// TIA Portal project "practical4 simba chipsFINAL" (V16)

(* hardware
DEVICE "S7300/ET200M station_1"  S7-300 station
   slot 0: "Rail_0"  Rail  6ES7 390-1***0-0AA0
   slot 1: "PS 307 2A_1"  PS 307 2A  6ES7 307-1BA01-0AA0
   slot 2: "PLC_1"  CPU 314C-2 DP  6ES7 314-6CH04-0AB0  V3.3
      slot 0: "MPI interface_1"  MPI
      slot 1: "DP interface_1"  DP
      slot 2: "DI 24/DO 16_1"  DI24/DO16
      slot 3: "AI 5/AO 2_1"  AI5/AO2
      slot 4: "Count_1"  Counter
      slot 5: "Positioning_1"  Positioning
DEVICE "HMI_1"  KTP700 Basic DP
   slot 0: "HMI_1"  KTP700 Basic DP  6AV2 123-2GA03-0AX0  16.0.0.0
   slot 1: "HMI_RT_1"  KTP700 Basic DP  6AV2 123-2GA03-0AX0  16.0.0.0
   slot 7: "HMI_1.MPI/DP_CP_1"  MPI/DP Interface  16.0.0.0
*)

// ===== PLC "PLC_1"  CPU 314C-2 DP =====

VAR_GLOBAL   // PLC tag table "Default tag table"
   "START" AT %M0.0 : Bool;
   "STOP" AT %M0.1 : Bool;
   "CONVEYOR 4" AT %Q0.0 : Bool;
   "RUNMODE" AT %Q1.3 : Bool;
   "OIL HEATER" AT %Q0.1 : Bool;
   "OIL HEATER TIMER" AT %T0 : Timer;
   "HEATER OUTPUT" AT %Q0.2 : Bool;
   "CONVEYOR 1" AT %Q0.3 : Bool;
   "CUTTING MACHINE" AT %Q0.4 : Bool;
   "CONVEYOR 2" AT %Q0.5 : Bool;
   "FRYING MACHINE" AT %Q0.6 : Bool;
   "CHIPS FRIER" AT %T1 : Timer;
   "CONVEYOR 3" AT %Q0.7 : Bool;
   "SENSOR" AT %M0.3 : Bool;
   "CHIPS COUNTER" AT %C0 : Counter;
   "COUNTER OUTPUT" AT %Q1.0 : Bool;
   "RESET" AT %M0.4 : Bool;
   "MAX" AT %MW0 : Word;
   "LOADING DURATION" AT %Q1.1 : Bool;
   "LOADING TIMER" AT %T2 : Timer;
   "TRUCK" AT %Q1.2 : Bool;
   "DELAY CONVEYOR 2" AT %T3 : Timer;
   "COMPARATOR OUTPUT" AT %Q1.4 : Bool;
   "SET VALUE" AT %M0.5 : Bool;
END_VAR

ORGANIZATION_BLOCK "Main"   // OB1, LAD
TITLE = "Main Program Sweep (Cycle)"
{ S7_Optimized_Access := 'FALSE' }
VERSION : 0.1
   VAR_TEMP
      OB1_EV_CLASS : Byte;   // Bits 0-3 = 1 (Coming event), Bits 4-7 = 1 (Event class 1)
      OB1_SCAN_1 : Byte;   // 1 (Cold restart scan 1 of OB 1), 3 (Scan 2-n of OB 1)
      OB1_PRIORITY : Byte;   // Priority of OB Execution
      OB1_OB_NUMBR : Byte;   // 1 (Organization block 1, OB1)
      OB1_RESERVED_1 : Byte;   // Reserved for system
      OB1_RESERVED_2 : Byte;   // Reserved for system
      OB1_PREV_CYCLE : Int;   // Cycle time of previous OB1 scan (milliseconds)
      OB1_MIN_CYCLE : Int;   // Minimum cycle time of OB1 (milliseconds)
      OB1_MAX_CYCLE : Int;   // Maximum cycle time of OB1 (milliseconds)
      OB1_DATE_TIME : Date_And_Time;   // Date and time OB1 started
   END_VAR
   VAR_TEMP   // added for the SCL form of the ladder/FBD networks
      _w1 : Bool;
      _s5time1 : S5Time;
   END_VAR
BEGIN

REGION Network 1: LATCHING CIRCUIT
   // Start button activates the system, Stop button deactivates the system. Runnmode is used as holding switch.
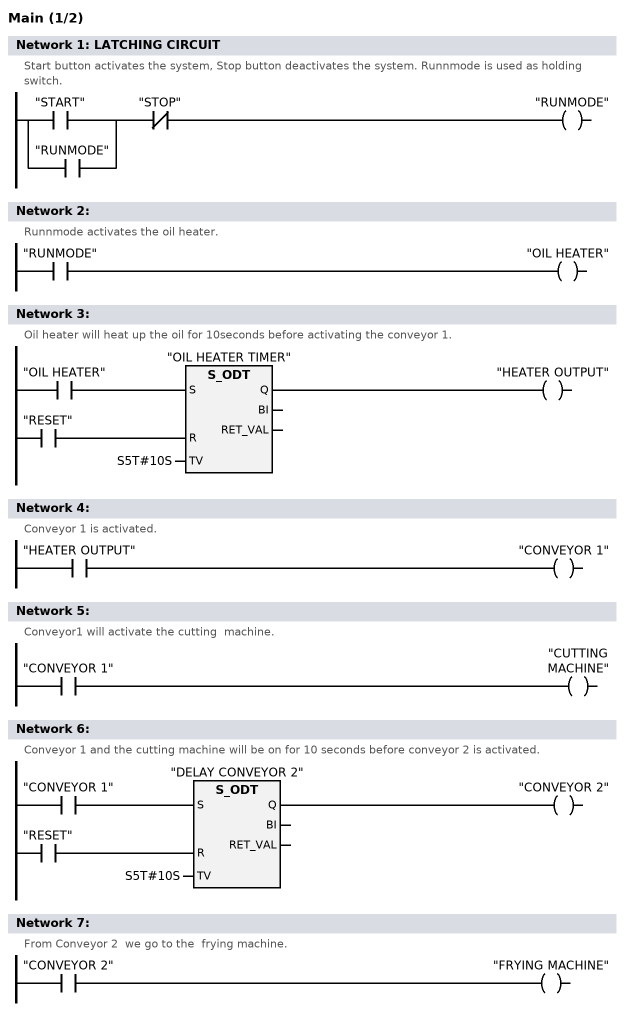
   RUNG wire#powerrail
      Contact( "START" )
      wire#w1
      I_Contact( "STOP" )
      Coil( "RUNMODE" )
   END_RUNG
   RUNG wire#powerrail
      Contact( "RUNMODE" )
   END_RUNG wire#w1
   // the same network as SCL:
   "RUNMODE" := ("START" OR "RUNMODE") AND NOT "STOP";
END_REGION

REGION Network 2
   // Runnmode activates the oil heater.
   RUNG wire#powerrail
      Contact( "RUNMODE" )
      Coil( "OIL HEATER" )
   END_RUNG
   // the same network as SCL:
   "OIL HEATER" := "RUNMODE";
END_REGION

REGION Network 3
   // Oil heater will heat up the oil for 10seconds before activating the conveyor 1.
   RUNG wire#powerrail
      Contact( "OIL HEATER" )
      S_ODT(T_NO := "OIL HEATER TIMER", R := wire#w1, TV := S5T#10S, BI =>, RET_VAL =>)
      Coil( "HEATER OUTPUT" )
   END_RUNG
   RUNG wire#powerrail
      Contact( "RESET" )
   END_RUNG wire#w1
   // the same network as SCL:
   #_s5time1 := S_ODT(T_NO := "OIL HEATER TIMER", S := "OIL HEATER", R := "RESET", TV := S5T#10S, Q => #_w1);
   "HEATER OUTPUT" := #_w1;
END_REGION

REGION Network 4
   // Conveyor 1 is activated.
   RUNG wire#powerrail
      Contact( "HEATER OUTPUT" )
      Coil( "CONVEYOR 1" )
   END_RUNG
   // the same network as SCL:
   "CONVEYOR 1" := "HEATER OUTPUT";
END_REGION

REGION Network 5
   // Conveyor1 will activate the cutting  machine.
   RUNG wire#powerrail
      Contact( "CONVEYOR 1" )
      Coil( "CUTTING MACHINE" )
   END_RUNG
   // the same network as SCL:
   "CUTTING MACHINE" := "CONVEYOR 1";
END_REGION

REGION Network 6
   // Conveyor 1 and the cutting machine will be on for 10 seconds before conveyor 2 is activated.
   RUNG wire#powerrail
      Contact( "CONVEYOR 1" )
      S_ODT(T_NO := "DELAY CONVEYOR 2", R := wire#w1, TV := S5T#10S, BI =>, RET_VAL =>)
      Coil( "CONVEYOR 2" )
   END_RUNG
   RUNG wire#powerrail
      Contact( "RESET" )
   END_RUNG wire#w1
   // the same network as SCL:
   #_s5time1 := S_ODT(T_NO := "DELAY CONVEYOR 2", S := "CONVEYOR 1", R := "RESET", TV := S5T#10S, Q => #_w1);
   "CONVEYOR 2" := #_w1;
END_REGION

REGION Network 7
   // From Conveyor 2  we go to the  frying machine.
   RUNG wire#powerrail
      Contact( "CONVEYOR 2" )
      Coil( "FRYING MACHINE" )
   END_RUNG
   // the same network as SCL:
   "FRYING MACHINE" := "CONVEYOR 2";
END_REGION

REGION Network 8
   // Frying machine will fry the chips for 20 seconds  before transporting  the chips via conveyor 3 to the boxes.
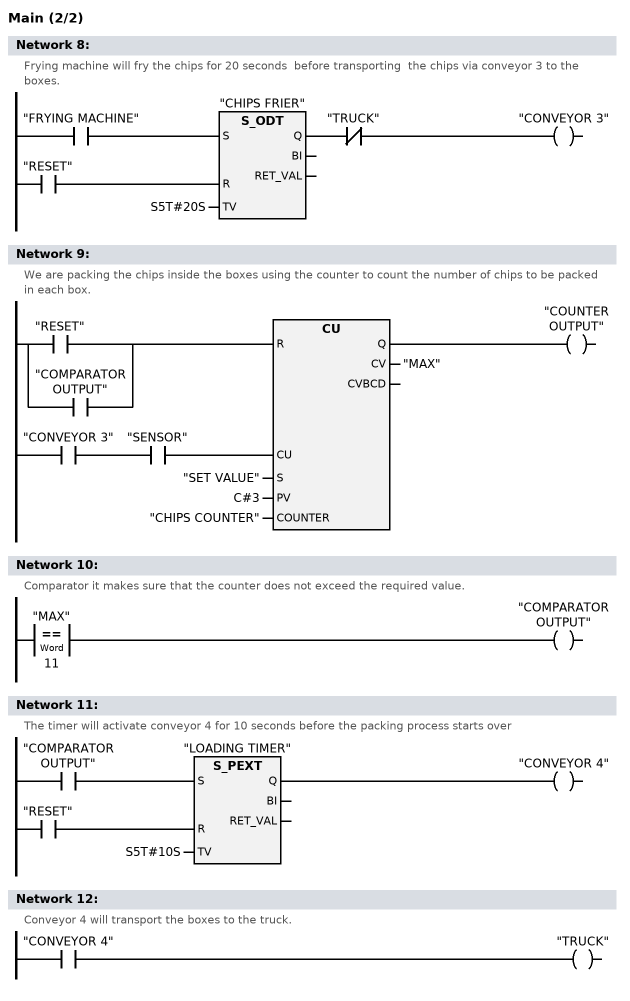
   RUNG wire#powerrail
      Contact( "FRYING MACHINE" )
      S_ODT(T_NO := "CHIPS FRIER", R := wire#w1, TV := S5T#20S, BI =>, RET_VAL =>)
      I_Contact( "TRUCK" )
      Coil( "CONVEYOR 3" )
   END_RUNG
   RUNG wire#powerrail
      Contact( "RESET" )
   END_RUNG wire#w1
   // the same network as SCL:
   #_s5time1 := S_ODT(T_NO := "CHIPS FRIER", S := "FRYING MACHINE", R := "RESET", TV := S5T#20S, Q => #_w1);
   "CONVEYOR 3" := #_w1 AND NOT "TRUCK";
END_REGION

REGION Network 9
   // We are packing the chips inside the boxes using the counter to count the number of chips to be packed  in each box.
   // no SCL statement known for Cu: written as a call
   Cu(cu := "CONVEYOR 3" AND "SENSOR",
      r := "RESET" OR "COMPARATOR OUTPUT",
      s := "SET VALUE",
      pv := C#3,
      "counter" := "CHIPS COUNTER",
      q => #_w1,
      cv => "MAX");
   "COUNTER OUTPUT" := #_w1;
END_REGION

REGION Network 10
   // Comparator it makes sure that the counter does not exceed the required value.
   RUNG wire#powerrail
      { S7_Templates := "SrcType := Word" } EQ_Contact(in1 := "MAX", in2 := 11)
      Coil( "COMPARATOR OUTPUT" )
   END_RUNG
   // the same network as SCL:
   "COMPARATOR OUTPUT" := "MAX" = 11;
END_REGION

REGION Network 11
   // The timer will activate conveyor 4 for 10 seconds before the packing process starts over
   RUNG wire#powerrail
      Contact( "COMPARATOR OUTPUT" )
      S_PEXT(T_NO := "LOADING TIMER", R := wire#w1, TV := S5T#10S, BI =>, RET_VAL =>)
      Coil( "CONVEYOR 4" )
   END_RUNG
   RUNG wire#powerrail
      Contact( "RESET" )
   END_RUNG wire#w1
   // the same network as SCL:
   #_s5time1 := S_PEXT(T_NO := "LOADING TIMER",
                       S := "COMPARATOR OUTPUT",
                       R := "RESET",
                       TV := S5T#10S,
                       Q => #_w1);
   "CONVEYOR 4" := #_w1;
END_REGION

REGION Network 12
   // Conveyor 4 will transport the boxes to the truck.
   RUNG wire#powerrail
      Contact( "CONVEYOR 4" )
      Coil( "TRUCK" )
   END_RUNG
   // the same network as SCL:
   "TRUCK" := "CONVEYOR 4";
END_REGION
END_ORGANIZATION_BLOCK

(* ===== HMI "HMI_RT_1" =====
system functions are stored by id; their names below are inferred from use
connection "HMI_Connection_1": IF1 B, SIMATIC S7 300/400 MPI

HMI tags "Default tag table"
   "Tag_ScreenNumber" : UInt, internal
   "START" : Bool = PLC START AT %M0.0, 1 s
   "STOP" : Bool = PLC STOP AT %M0.1, 1 s
   "SENSOR" : Bool = PLC SENSOR AT %M0.3, 1 s
   "OIL HEATER" : Bool = PLC "OIL HEATER" AT %Q0.1, 1 s
   "HEATER OUTPUT" : Bool = PLC "HEATER OUTPUT" AT %Q0.2, 1 s
   "CONVEYOR 2" : Bool = PLC "CONVEYOR 2" AT %Q0.5, 1 s
   "CONVEYOR 1" : Bool = PLC "CONVEYOR 1" AT %Q0.3, 1 s
   "CUTTING MACHINE" : Bool = PLC "CUTTING MACHINE" AT %Q0.4, 1 s
   "OIL HEATER TIMER" : Timer = PLC "OIL HEATER TIMER" AT %T0, 1 s
   "RUNMODE" : Bool = PLC RUNMODE AT %Q1.3, 1 s
   "DELAY CONVEYOR 2" : Timer = PLC "DELAY CONVEYOR 2" AT %T3, 1 s
   "CONVEYOR 3" : Bool = PLC "CONVEYOR 3" AT %Q0.7, 1 s
   "FRYING MACHINE" : Bool = PLC "FRYING MACHINE" AT %Q0.6, 1 s
   "COUNTER OUTPUT" : Bool = PLC "COUNTER OUTPUT" AT %Q1.0, 1 s
   "CHIPS FRIER" : Timer = PLC "CHIPS FRIER" AT %T1, 1 s
   "CHIPS COUNTER" : Counter = PLC "CHIPS COUNTER" AT %C0, 1 s
   "CONVEYOR 4" : Bool = PLC "CONVEYOR 4" AT %Q0.0, 1 s
   "movement" : Int, internal
   "LOADING DURATION" : Bool = PLC "LOADING DURATION" AT %Q1.1, 1 s
   "LOADING TIMER" : Timer = PLC "LOADING TIMER" AT %T2, 1 s
   "RESET" : Bool = PLC RESET AT %M0.4, 1 s

Template "Template_1" 800x480
   SymbolicIOField "Symbolic_IO_Field_Screen" at 93,9 size 600x33; TextOff '0'; TextOn '1'; TextList "TextList_ScreenNames"
      ProcessValue <- "Tag_ScreenNumber"
      on Change: ActivateScreenByNumber("Tag_ScreenNumber", 0)
   DateTimeField "HmiScreenItemData" at 695,25 size 105x25
   DateTimeField "HmiScreenItemData_1" at 695,0 size 105x25
   GraphicView "Logo" at 0,0 size 91x51; Picture "Logo of HMI_1"

screen "Root screen" 800x480, template "Template_1"
   on GenerateScreen: function_f9c01323("movement", 1, 100, 0, 1)
   TextField "HmiScreenItemData" at 43,19 size 640x25; Text 'Welcome to HMI_1 (KTP700 Basic+ DP)!'
   Button "Button_1" at 681,72 size 96x32; TextOff 'START'
      on Press: SetBit("START")
      on Release: ResetBit("START")
   Button "Button_2" at 681,120 size 96x32; TextOff 'STOP'
      on Press: SetBit("STOP")
      on Release: ResetBit("STOP")
   GraphicView "Graphic view_2" at 303,276 size 366x43; Picture "Graphic_2"
   GraphicView "Graphic view_7" at 363,196 size 60x66; Picture "Graphic_13"
   GraphicView "Graphic view_8" at 572,307 size 188x90; Picture "Graphic_16"
   Rectangle "Rectangle_1" at 608,356 size 30x26
      Appearance <- "OIL HEATER"
   Rectangle "Rectangle_4" at 381,198 size 22x22
      Appearance <- "CUTTING MACHINE"
   IOField "I/O field_1" at 28,57 size 96x32; FormatPattern 99999
      Appearance <- "OIL HEATER TIMER"
      ProcessValue <- "OIL HEATER TIMER"
   IOField "I/O field_2" at 416,57 size 96x32; FormatPattern 999999
      ProcessValue <- "CHIPS FRIER"
   TextField "Text field_1" at 28,87 size 84x23; Text 'oil heater'
   IOField "I/O field_3" at 216,57 size 96x32; FormatPattern 99999
      ProcessValue <- "DELAY CONVEYOR 2"
   TextField "Text field_2" at 412,89 size 86x23; Text 'chips frier'
   TextField "Text field_3" at 193,89 size 130x23; Text 'Conveyor delay'
   Button "Button_5" at 680,207 size 99x32; TextOff 'SCREEN_1'; TextOn 'Screen_3'
      on Click: ActivateScreen("Screen_3", 0)
   Button "Button_4" at 678,257 size 99x32; TextOff 'Screen_2'; TextOn 'Screen_4'
      on Click: ActivateScreen("Screen_4", 0)
   Button "Button_6" at 683,164 size 96x32; TextOff 'RESET'
      Appearance <- "RESET"
      on Press: SetBit("RESET")
      on Release: ResetBit("RESET")
   GraphicView "Graphic view_1" at 110,179 size 285x41; Picture "Graphic_21"
      Appearance <- "CONVEYOR 1"
   GraphicView "Graphic view_3" at 303,319 size 131x78; Picture "Graphic_22"
   Rectangle "Rectangle_2" at 327,332 size 42x37
      Appearance <- "CONVEYOR 2"
   GraphicView "Graphic view_4" at 13,370 size 116x73; Picture "Graphic_22"
   Rectangle "Rectangle_3" at 35,378 size 42x37
      Appearance <- "CONVEYOR 1"
   GraphicView "Graphic view_5" at 0,199 size 134x179; Picture "Graphic_23"

screen "Screen_3" 800x480
   on GenerateScreen: function_f9c01323("movement", 1, 100, 0, 1)
   GraphicView "Graphic view_8" at 15,19 size 185x83; Picture "Graphic_16"
   GraphicView "Graphic view_2" at 128,111 size 427x45; Picture "Graphic_2"
      Appearance <- "COUNTER OUTPUT"
   Button "Button_3" at 650,57 size 137x32; TextOff 'COUNTER UP'
      on Release: ResetBit("SENSOR")
      on Press: SetBit("SENSOR")
   Rectangle "Rectangle_2" at 50,62 size 35x27
      Appearance <- "FRYING MACHINE"
   GraphicView "Graphic view_1" at 516,139 size 64x84; Picture "Graphic_4"
   GraphicView "Graphic view_4" at 487,234 size 125x106; Picture "Graphic_17"
   Rectangle "Rectangle_3" at 528,144 size 27x31
      Appearance <- "COUNTER OUTPUT"
   IOField "I/O field_1" at 441,168 size 65x31; FormatPattern 9
      ProcessValue <- "CHIPS COUNTER"
   Button "Button_2" at 651,168 size 136x32; TextOff 'HOME_SCREEN'; TextOn 'Root screen'
      on Click: ActivateScreen("Root screen", 0)
   Button "Button_1" at 651,107 size 137x32; TextOff 'Screen_2'; TextOn 'Screen_4'
      on Click: ActivateScreen("Screen_4", 0)
   GraphicView "Graphic view_5" at 128,153 size 131x78; Picture "Graphic_22"
   Rectangle "Rectangle_1" at 158,163 size 42x37
      Appearance <- "CONVEYOR 3"
   IOField "I/O field_2" at 241,4 size 96x32; FormatPattern 999999
      ProcessValue <- "CHIPS FRIER"
   TextField "Text field_2" at 237,34 size 86x23; Text 'chips frier'

screen "Screen_4" 800x480
   on GenerateScreen: function_f9c01323("movement", 1, 100, 0, 1)
   GraphicView "Graphic view_1" at 224,67 size 64x84; Picture "Graphic_4"
   GraphicView "Graphic view_2" at 172,246 size 420x47; Picture "Graphic_2"
      Appearance <- "CONVEYOR 4"
   Rectangle "Rectangle_3" at 232,74 size 27x31
      Appearance <- "COUNTER OUTPUT"
   IOField "I/O field_1" at 125,85 size 65x31; FormatPattern 9
      ProcessValue <- "CHIPS COUNTER"
   Button "Button_3" at 662,79 size 130x32; TextOff 'COUNTER UP'
      on Release: ResetBit("SENSOR")
      on Press: SetBit("SENSOR")
   Button "Button_2" at 663,189 size 137x32; TextOn 'Root screen'; TextOff 'HOME_SCREEN'
      on Click: ActivateScreen("Root screen", 0)
   Button "Button_1" at 663,133 size 133x32; TextOff 'Screen_1'; TextOn 'Screen_3'
      on Click: ActivateScreen("Screen_3", 0)
   GraphicView "Graphic view_5" at 205,177 size 116x97; Picture "Graphic_18"
      Visibility <- "CONVEYOR 4"
      HorizontalMovement <- "movement"
   GraphicView "Graphic view_4" at 204,177 size 117x97; Picture "Graphic_19"
      Visibility <- "CONVEYOR 4"
   GraphicView "Graphic view_3" at 190,290 size 131x78; Picture "Graphic_22"
   Rectangle "Rectangle_1" at 224,301 size 42x37
      Appearance <- "CONVEYOR 4"
*)